TYPE U_TOUCH_PROBE_STATE :
UNION
  stState              : ARRAY[1..MAX_TOUCH_PROBE] OF ST_STATE_TOUCH_PROBE;

  byState    AT %i*   : ARRAY[1..MAX_TOUCH_PROBE] OF
                        ARRAY[1..SIZEOF(ST_STATE_TOUCH_PROBE)] OF BYTE;
END_UNION
END_TYPE

(* stored: Version 1.1.0.1
   DUT U_TOUCH_PROBE_STATE: Id {8da8cfa8-e95e-423a-bb11-2e411f04dfaa} *)
